Yaskawa INFORM job: position_test.JBI

/JOB
//NAME POS_TEST
//POS
///NPOS 1,0,1,0,0,0
///TOOL 0
///POSTYPE BASE
///RECTAN
///RCONF 1,0,0,0,0,0,0,0,0,0,0,0,0,0,0,0,0,0,0,0,0,0,0,0
C00000=2000.000,0.000,0.000,-90.0000,0.0000,-90.0000
///POSTYPE PULSE
///PULSE
EC00000=0
//INST
///DATE 2022/12/28 11:56
///ATTR SC,RW,RJ
////FRAME BASE
///GROUP1 RB1,ST1
NOP
MOVJ C00000 EC00000 VJ=15.00
END
